Universal Robots PolyScope program: TM0512_rs3demo_Ratchet.urp

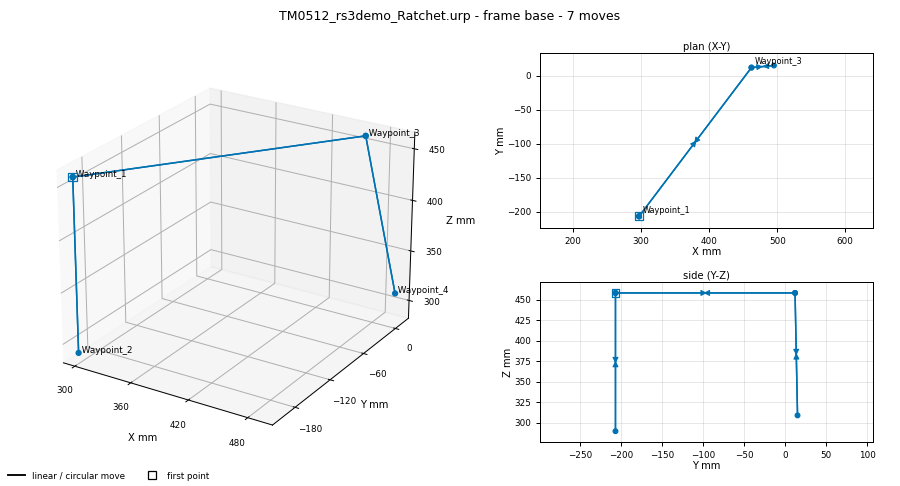
[picture p0: tool path of TM0512_rs3demo_Ratchet.urp in frame base, 7 of 7 moves have a stored position in this frame; points joined in program order, loops and branches not executed]
Program TM0512_rs3demo_Ratchet (installation=default directory=/programs createdIn=5.11.9.1010452 lastSavedIn=5.11.9.1010452 robotSerialNumber=20225200364)
Calibrated DH parameters: a=[0.00002, -0.569483, -0.54992, -0.00001, -0.000036, 0]; d=[0.180894, -146.691669, 192.918669, -46.053088, 0.119778, 0.115602]; alpha=[1.571425, -0.001534, 0.003359, 1.568739, -1.571477, 0]; deltaTheta=[0, 0.376258, -0.101074, -0.275185, -0.000002, 0]
Robot Program (runOnlyOnce=false)
  MoveL speed 50 mm/s, acceleration 1200 mm/s^2 (useActiveTCP=true) feature=Base
    Waypoint Waypoint_1: TCP in base x=296.88 y=-206.693 z=458.109 mm, rx=2.2142 ry=-2.1954 rz=0.0213 rad; joints [-5.52, -53.173, -136.663, -80.366, 88.693, -6.097] deg
    URCap RG Grip (OnRobot, OnRobot A/S) dataModel(rg-target-force=40.0, rg-target-width=0.1, Variable(key=on_return, variable(name=on_return)))
    Waypoint Waypoint_2: TCP in base x=296.936 y=-206.697 z=289.73 mm, rx=2.2142 ry=-2.1955 rz=0.0214 rad; joints [-5.536, -63.214, -151.137, -55.849, 88.676, -6.018] deg
    URCap RG Grip (OnRobot, OnRobot A/S) dataModel(rg-target-force=40.0, rg-target-width=0.075)
    Waypoint Waypoint_1: TCP in base x=296.88 y=-206.693 z=458.109 mm, rx=2.2142 ry=-2.1954 rz=0.0213 rad; joints [-5.52, -53.173, -136.663, -80.366, 88.693, -6.097] deg
    Waypoint Waypoint_3: TCP in base x=462.084 y=11.994 z=458.103 mm, rx=2.214 ry=-2.1955 rz=0.0213 rad; joints [23.916, -67.328, -130.079, -73.521, 88.999, 23.392] deg
    Waypoint Waypoint_4: TCP in base x=495.146 y=15.008 z=308.979 mm, rx=2.2142 ry=-2.1954 rz=0.0215 rad; joints [22.58, -80.616, -138.326, -51.956, 88.943, 22.129] deg
    URCap RG Grip (OnRobot, OnRobot A/S) dataModel(rg-target-force=40.0, rg-target-width=0.1)
    Waypoint Waypoint_3: TCP in base x=462.084 y=11.994 z=458.103 mm, rx=2.214 ry=-2.1955 rz=0.0213 rad; joints [23.916, -67.328, -130.079, -73.521, 88.999, 23.392] deg
    Waypoint Waypoint_1: TCP in base x=296.88 y=-206.693 z=458.109 mm, rx=2.2142 ry=-2.1954 rz=0.0213 rad; joints [-5.52, -53.173, -136.663, -80.366, 88.693, -6.097] deg
    Halt
